TYPE ST_SettingsLiftingTransport :
STRUCT
	//Lift
	stLiftSpeedProfileJogging : ST_SpeedProfile;
	stLiftSpeedProfilePositioning : ST_SpeedProfile;   
	arr_LiftPositioningProfile : ARRAY[0..10] OF ST_PositioningProfile;
	
	//Transport
	stTransportSpeedProfileJogging : ST_SpeedProfile;
	stTransportSpeedProfilePositioning : ST_SpeedProfile;
	arr_TransportPositioningProfile : ARRAY[0..5] OF ST_PositioningProfile;
END_STRUCT
END_TYPE

(* stored: Version 1.1.0.1, ProductVersion 3.1.4024.12
   DUT ST_SettingsLiftingTransport: Id {cad671c8-daf9-4539-9908-38693c7e494e} *)
